PROGRAM MAIN
VAR
END_VAR

END_PROGRAM

(* stored: Version 1.1.0.1
   POU MAIN: Id {dcf86679-b5e8-4481-bba3-406704c5d86b} *)
